INTERFACE I_Datatype extends I_Serializable, I_Deserializable, I_Disposable

METHOD PUBLIC Accept
VAR_INPUT
	Visitor : I_DatatypeVisitor;
END_VAR
END_METHOD

PROPERTY PUBLIC Address : PVOID
GET
END_GET
END_PROPERTY

METHOD PUBLIC ClearReference
VAR_INPUT
END_VAR
END_METHOD

METHOD Clone : I_Datatype
END_METHOD

PROPERTY PUBLIC IsUserDefined : BOOL
GET
END_GET
END_PROPERTY

METHOD PUBLIC SerializeTypeWith
VAR_INPUT
	Serializer : I_Serializer;
END_VAR
END_METHOD

PROPERTY PUBLIC Size : UDINT
GET
END_GET
END_PROPERTY

METHOD PUBLIC TryCopyFrom : BOOL
VAR_INPUT
	Source : I_Datatype;
END_VAR
END_METHOD

METHOD PUBLIC ABSTRACT TryDeserializeFrom : BOOL
VAR_INPUT
	Deserializer : I_Deserializer;
	Feedback : I_DeserializerFeedback;
END_VAR
END_METHOD

METHOD TryMakeReferenceTo : BOOL
VAR_INPUT
	Target : I_Datatype;
END_VAR
END_METHOD

METHOD PUBLIC TryResolveAsAliasDatatype : BOOL
VAR_INPUT
	Destination : REFERENCE TO I_AliasDatatype;
END_VAR
END_METHOD

METHOD PUBLIC TryResolveAsEnumDatatype : BOOL
VAR_INPUT
	Destination : REFERENCE TO I_EnumDatatype;
END_VAR
END_METHOD

METHOD PUBLIC TryResolveAsStructuredDatatype : BOOL
VAR_INPUT
	Destination : REFERENCE TO I_StructuredDatatype;
END_VAR
END_METHOD

PROPERTY PUBLIC TypeName : T_MAXSTRING
GET
END_GET
END_PROPERTY

END_INTERFACE

(* stored: Version 1.1.0.1, ProductVersion 3.1.4024.12
   Itf I_Datatype: Id {f9228532-ea06-0cea-156b-b78f9ec3688c}
   Method Accept: Id {222f1d5c-17b7-0656-3c13-c8636228d76a}
   Property Address: Id {208dfa1e-f2c9-0ae5-2623-d0ed741ef8b5}
   Get Get: Id {54c60cea-06d9-0436-2d98-e11a2955b4ed}
   Method ClearReference: Id {3e6f425d-2cc3-0286-2773-4d68f68355c3}
   Method Clone: Id {cba15b80-9b6c-09f2-371d-4de2af359262}
   Property IsUserDefined: Id {acc2d798-2f2b-47aa-b664-a7dabd1fa5e5}
   Get Get: Id {98703baf-5563-449d-9176-64070ab24cd7}
   Method SerializeTypeWith: Id {49c39a8f-18b1-0e61-0283-6c14f52574e5}
   Property Size: Id {82556afa-6c09-02a5-21b3-c6f1b10f4d7a}
   Get Get: Id {a604ab4c-7ad4-0419-3fa1-ddd96273706f}
   Method TryCopyFrom: Id {799ca117-6aed-4029-8900-4a8b83228335}
   Method TryDeserializeFrom: Id {37f3fe44-520f-0d11-174b-facb5919c405}
   Method TryMakeReferenceTo: Id {71e1f5db-87ba-0edb-12be-d38f86ff6c6e}
   Method TryResolveAsAliasDatatype: Id {6901fdc3-b8df-0a50-076a-29e0627543a7}
   Method TryResolveAsEnumDatatype: Id {e7be0424-a479-0a55-1293-36f08e36456b}
   Method TryResolveAsStructuredDatatype: Id {1f72b16a-4b89-0abc-267a-2a1e1af6e054}
   Property TypeName: Id {ea4da69c-fd1b-0766-085e-ae11be47eeb6}
   Get Get: Id {8d4b7908-183b-02d9-27cf-9fb0bce53892} *)
